{attribute addProperty BoxType "EK1110-0043-0016"}
{attribute addProperty Id "InfoDataInfoData_192954DE162"}
{attribute addProperty CRC "395970889"}
{attribute addProperty SizeInBites "16"}
{attribute addProperty SizeInBytes "2"}
TYPE EK1110_179A0949 :
STRUCT
	{attribute addProperty Name "InfoData"}
	InfoData : InfoData_192954DE;
END_STRUCT
END_TYPE

(* stored: Version 1.2.0.0, ProductVersion 3.1.4024.9
   DUT EK1110_179A0949: Id {080461fe-aa32-4cdb-8328-6787be0b1961} *)
